(* CoDeSys 2.3.9.42 project: 2_poz_reg_97.pro *)
(* Libraries: standard.lib 4.10.05 11:14:46, Util.lib 18.5.10 15:14:28 *)

(* POU PLC_PRG, CFC *)
PROGRAM PLC_PRG
VAR
	rs_1: RS;
		ustavka: REAL;
	tek_Temperatura: REAL;
	Ten_on: BOOL;
END_VAR
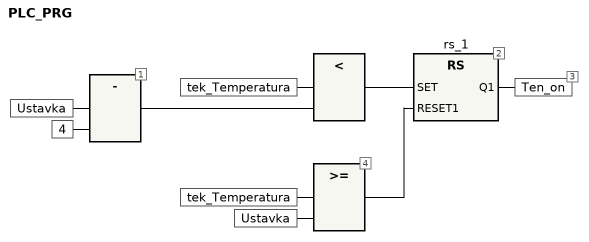
_CFC_ (* Continuous Function Chart, elements in execution order *)
#0 <(tek_Temperatura, #1)
#1 -(Ustavka, 4)
#2 rs_1:RS(SET: #0, RESET1: #4)
#3 Ten_on <= #2.Q1
#4 >=(tek_Temperatura, Ustavka)
_END_CFC_
END_PROGRAM
